(* PLC project maintained_button, Dassault Systèmes ControlBuild 2024x *)
(* stored: creationDateTime 2023-10-03T11:13:21-01:00 *)

(* This module simulates a maintained contact push button. *)
FUNCTION_BLOCK equipment_library.maintained_button
  VAR_OUTPUT
    pb : BOOL := false;
  END_VAR
  VAR
    action : BOOL := false;
  END_VAR
  VAR CONSTANT
    PBLogic : BOOL := true;
  END_VAR

(* -----------------------------------------------------------------	*)
(* Type : Model of Operative Behaviour					*)
(* Category :  Power								*)
(* Author : Dassault Systemes						*)
(* Update date : June 2018							*)
(* -----------------------------------------------------------------	*)
(* This module simulates a maintained contact push button. 		*)
(* -----------------------------------------------------------------	*)



pb := (action XOR NOT PBLogic);
END_FUNCTION_BLOCK
